(* PLC project Generated.project, CODESYS CODESYS V3.5 SP19 Patch 1 *)
(* stored: creationDateTime 2026-09-06T13:00:42.508254, modificationDateTime 2026-09-06T13:00:42.508254 *)

(* ═══════════════════════════════════════════════════════════════ ↔️ ST_TranslationHMI — Données d'échange IHM pour le Translation M3 ─────────────────────────────────────────────────────────────── 🎨 Destiné à l'affichage des états, commandes et diagnostics du translation. 📄 Structuration en Cmd / State / Safety / Bypass / Test — doc métier : DOC/AF/AF_Partie-11_Fonction_Translation_v2.3.md ═══════════════════════════════════════════════════════════════ *)
TYPE ST_TranslationHMI : STRUCT
  Cmd : ST_TranslationCmd;  (* 🎮 Commandes opérateur (manuel / maintenance) *)
  State : ST_TranslationState;  (* 🚦 États & diagnostics *)
  Cfg : ST_TranslationCfg;  (* Configurations et limites — champ Cfg manquait initialement (contrairement à ST_WinchHMI) *)
  Bypass : ST_BypassTranslation;  (* Bypass maintenance *)
  Safety : ST_SafetyTranslation;  (* 🛡️ Sécurité (FB_Safety_Translation) *)
END_STRUCT;
END_TYPE

(* ═══════════════════════════════════════════════════════════════ ST_BypassTranslation — Bypass maintenance dédiés à Translation M3 ─────────────────────────────────────────────────────────────── 🔒 Doctrine : actionnable UNIQUEMENT en MAINT_N2, RETAIN, jamais masque les autres défauts du même bloc (voir REGISTRE_ACTIONS_Bypass_v1.0 (archive)). ═══════════════════════════════════════════════════════════════ *)
TYPE ST_BypassTranslation : STRUCT
  OperatorComm : BOOL;  (* 📡 1. Communication & Systèmes auxiliaires 📡 Bypass communication esclave CANopen Joystick / heartbeat IHM *)
  DriveComm : BOOL;  (* 📡 Bypass diagnostic esclave EtherCAT AC600 (variateur) *)
  ContactorFeedback : BOOL;  (* 🔌 Bypass feedbacks contacteur de frein *)
  PhaseRotation : BOOL;  (* ⚡ Bypass défaut rotation de phases (commun machine) *)
  BrakeThermal : BOOL;  (* 🌡️ Bypass surchauffe thermique frein (commun machine) *)
  LimitSwitch : BOOL;  (* 🚧 2. Limites physiques et Positionnement 🚧 Bypass fins de course physiques avant/arrière *)
  SensorIncoherent : BOOL;  (* 🧭 Bypass incohérence mot capteurs de position *)
  MinHeight : BOOL;  (* : Bypass interlock hauteur mini M1/M2 requise pour translation *)
  MecaA : BOOL;  (* ⚙️ 3. Sécurité Mécanique (Méca A-B) 🔄 Bypass Méca A : mouvement non commandé à l'arrêt *)
  MecaB : BOOL;  (* 🛑 Bypass Méca B : absence confirmation arrêt (frein/contacteurs) *)
  Safety : BOOL;  (* 🛡️ 4. Hiérarchie & Restauration 🛡️ Bypass groupé : tous les bits qui provoquent un PowerCutOff *)
  Process : BOOL;  (* ⚙️ Bypass groupé : tous les bits qui provoquent un SafeStop *)
  Global : BOOL;  (* 🌐 Bypass Global : ignore toutes les sécurités de cet axe *)
  Initialized : BOOL := FALSE;  (* Flag restauration boot dédié (défaut FALSE non ambigu, contrairement à une valeur métier) 🚦 TRUE = bypass restauré depuis GVL_BypassRetain ce boot *)
END_STRUCT;
END_TYPE

(* ═══════════════════════════════════════════════════════════════ 🛡️ ST_SafetyTranslation — Diagnostics de sécurité pour la Translation M3 ─────────────────────────────────────────────────────────────── 🎨 Destiné à l'affichage des défauts de sécurité du translation. ═══════════════════════════════════════════════════════════════ *)
TYPE ST_SafetyTranslation : STRUCT
  Error : BOOL;  (* 🛡️ Bloc sécurité (Safety) en défaut *)
  ErrorId : WORD;  (* ❌ Code bitfield du défaut de sécurité (vue LIVE) *)
  LatchedId : WORD;  (* 🕘 Vue LATCHÉE : ErrorId figé au défaut, effacé au Reset (marqueur [HISTO]) *)
  ErrorOperatorComm : BOOL;  (* 🎮 Perte communication opérateur : joystick CAN ou heartbeat IHM (bit0) *)
  ErrorDriveComm : BOOL;  (* 📡 Perte communication EtherCAT variateur (bit1) *)
  ErrorPhaseRotation : BOOL;  (* ⚡ Mauvaise rotation de phases électriques (bit2) *)
  ErrorBrakeThermal : BOOL;  (* 🌡️ Surchauffe thermique frein commun (bit3) *)
  ErrorMecaB : BOOL;  (* 🛑 Absence confirmation arrêt (Méca B - bit4) *)
  ErrorMecaA : BOOL;  (* 🔄 Mouvement non commandé (Méca A - bit5) *)
  ErrorLimitSwitch : BOOL;  (* 🚧 Limite extrême Translation atteinte (bit6) *)
  ErrorSensorIncoherent : BOOL;  (* 🧭 Mot capteurs M3 incohérent (bit7) *)
  SafeStop : BOOL;  (* 🛡️ Décélération de sécurité demandée *)
  PowerCutOff : BOOL;  (* 🧨 Coupure puissance demandée *)
  EffectivePermitM3_Tremie : BOOL;  (* 🟢 Permis canonique M3 vers Trémie, TRUE = autorisé *)
  EffectivePermitM3_Maintenance : BOOL;  (* 🟢 Permis canonique M3 vers Maintenance/P1, TRUE = autorisé *)
  BlockedBySafety : BOOL;  (* 🚫 Synthèse globale : translation bloquée par la sécurité *)
  PowerCutOffSafety : BOOL;  (* 🧨 Synthèse sécurités critiques entraînant une coupure puissance *)
  SafeStopSafety : BOOL;  (* 🛡️ Synthèse défauts entraînant un SafeStop / Rampe rapide *)
END_STRUCT;
END_TYPE

(* ═══════════════════════════════════════════════════════════════ ST_TranslationCfg — Configurations et paramètres réglables pour Translation M3 ─────────────────────────────────────────────────────────────── 🎨 Destiné au paramétrage depuis l'IHM (RETAIN) — même patron que ST_WinchCfg. 📄 Vitesses de ralentissement d'approche réglables depuis l'IHM (RETAIN), même patron que ST_WinchCfg. ═══════════════════════════════════════════════════════════════ *)
TYPE ST_TranslationCfg : STRUCT
  CfgApproachSpeedTremie_Hz : REAL := 20;  (* 🐢 Vitesse réduite d'approche Trémie (Hz), déclenchée par capteur PV, Direction=1 — reglage nominal confirme operateur *)
  CfgApproachSpeedMaintenance_Hz : REAL := 20;  (* 🐢 Vitesse réduite d'approche Maintenance (Hz), déclenchée par capteur P1, Direction=-1 — reglage nominal confirme operateur *)
  CfgApproachSpeedP1_Hz : REAL := 20;  (* 🐢 Vitesse réduite d'approche P1 (Hz), déclenchée par capteur P2, Direction=-1 — reglage nominal confirme operateur *)
  Initialized : BOOL := FALSE;  (* Flag restauration boot (défaut FALSE non ambigu) — même patron que ST_WinchCfg 🚦 TRUE = config restaurée depuis GVL_PERSISTENT ce boot *)
END_STRUCT;
END_TYPE

(* ═══════════════════════════════════════════════════════════════ 🎮 ST_TranslationCmd — Commandes IHM pour la Translation M3 ─────────────────────────────────────────────────────────────── 🎨 Destiné au pilotage de la translation M3 depuis l'IHM. 📄 : Initialized protège SetFreq_Hz (seul réglage à survivre au reboot), sans pont générique pour ne jamais persister BtnTremie/BtnMaintenance. ═══════════════════════════════════════════════════════════════ *)
TYPE ST_TranslationCmd : STRUCT
  SelPositioning : BOOL;  (* 🎯 TRUE = positionneur sur SelTarget ; FALSE = jog libre *)
  SelTarget : INT;  (* 🔢 Numéro de la cible de position sélectionnée *)
  BtnTremie : BOOL;  (* ↔️ Requête marche vers Trémie (ex-BtnFwd), pilotage IHM exclusif *)
  BtnMaintenance : BOOL;  (* ↔️ Requête marche vers Maintenance (ex-BtnRev), pilotage IHM exclusif *)
  SetFreq_Hz : REAL;  (* 🎯 Consigne fréquence manuelle [Hz], limitée par PRG_06_Outputs *)
  InvertDirection : BOOL;  (* 🔀 Switch machine unique : GVL_IHM.Modes.Cmd.TglJoystickMaster (ST_ModesCmd), applicable à M1/M2 ET M3. 🔄 TRUE = inverse Fwd→Maintenance / Rev→Trémie (mise en service) *)
  TglMaintenanceZoneAccess : BOOL;  (* : autorisation CONSCIENTE zone Maintenance, EN PLUS de MAINT_N2 (Auth.MaintenanceM3TargetEnable) *)
  TglAllowWinchMoveAtTremie : BOOL;  (* T249 : autorisation CONSCIENTE montee/descente treuil couple (WinchSel=0) a la Tremie, EN PLUS de la garde WinchSel=2 forcee (FB_Modes) *)
  Initialized : BOOL := FALSE;  (* 🚦 TRUE = SetFreq_Hz restauré depuis GVL_PERSISTENT ce boot *)
  BtnSetAtP1 : BOOL;  (* 🎯 Forcage position P1 depuis IHM en MAINT_N2 (mise en service) *)
END_STRUCT;
END_TYPE

(* ═══════════════════════════════════════════════════════════════ 🚦 ST_TranslationState — États et retours IHM pour la Translation M3 ─────────────────────────────────────────────────────────────── 🎨 Destiné à l'affichage des retours et mesures de la translation M3. ═══════════════════════════════════════════════════════════════ *)
TYPE ST_TranslationState : STRUCT
  FBState : E_State;  (* 🚦 États & diagnostics FB_Translation 🤖 État de l'automate interne (FB_Translation) *)
  AxisBlockReason : E_TranslationTraceBlockReason;  (* 🧩 Cause prioritaire de blocage (miroir de TranslationTrace.BlockReason) *)
  Ready : BOOL;  (* 🟢 Translation prêt à fonctionner *)
  Busy : BOOL;  (* ⚙️ Mouvement en cours *)
  Done : BOOL;  (* ✅ Mouvement terminé avec succès *)
  Error : BOOL;  (* Translation en défaut *)
  ErrorId : WORD;  (* ❌ Code du défaut actif *)
  BrakeCmd : BOOL;  (* 🔓 Commande de desserrage du frein (lecture seule, TRUE = desserré) *)
  BrakeFeedback : BOOL;  (* 🔌 Retour physique direct : TRUE = frein OUVERT (desserré) *)
  PositionSensorTarget : BOOL;  (* 🎯 Capteur de détection de la position cible atteint *)
  PositionReached : BOOL;  (* ✅ Positionneur : cible sélectionnée atteinte (non mémorisé) *)
  DriveActualFreq_Hz : REAL;  (* 📈 Fréquence de sortie réelle du variateur (Hz) *)
  DriveControlWord : WORD;  (* ⚙️ Mot de commande AC600 réellement appliqué *)
  DriveFreqCmd_Hz : REAL;  (* 🎯 Commande fréquence réellement appliquée *)
  ActiveTremie : BOOL;  (* ↔️ Commande active vers Trémie *)
  ActiveMaintenance : BOOL;  (* ↔️ Commande active vers Maintenance *)
  SpeedCmd_Pct : REAL;  (* 📊 Commande active après arbitrage (0.0 à 100.0 %) *)
  FinalInterlockState : E_State;  (* 🛡️ État final lecture seule *)
  FinalInterlockReason : E_TranslationFinalInterlockReason;  (* 🛡️ Cause finale mémorisée *)
  FinalInterlockError : BOOL;  (* 🛡️ Défaut final mémorisé *)
  FinalInterlockErrorId : WORD;  (* 🛡️ Bitfield final *)
  BrakeCommandOpenConfirmed : BOOL;  (* 🔌 Contacteur/bobine desserrage confirmé, pas frein mécanique *)
  FinalBrakeTimeoutElapsed : TIME;  (* ⏱️ Écoulé watchdog 500ms *)
  DriveCommReady : BOOL;  (* 🔌 Diagnostic variateur EtherCAT (décodé — pas de bit-masking côté IHM) 📡 Variateur M3 : communication prête (StatusWord bit7) *)
  DrivePowerReady : BOOL;  (* ⚡ Variateur M3 : puissance prête (StatusWord bit0) *)
  PositionTremie : BOOL;  (* 📍 Mot capteurs et positions Translation M3 *)
  PositionPV : BOOL;
  PositionP2 : BOOL;
  PositionP1 : BOOL;
  PositionMaintenance : BOOL;
  AtTremie : BOOL;  (* : mot EXACT — front franc arrivée/cible (voir PositionXxx ci-dessus = cumulatif zone, réservé ralentissement) jeton "dernier capteur franchi" (front + libération sur mouvement confirmé) — logique de positionnement *)
  AtPV : BOOL;
  AtP2 : BOOL;
  AtP1 : BOOL;
  AtMaintenance : BOOL;
  M3StatusText : STRING(80);  (* T249-B : texte statut position M3 (INFO, lecture seule) — jeton "at position" sur front capteur sinon zone SensorsWord. Ex "M3 a P1 -> Maintenance", "M3 entre P2 et P1" *)
  EstimatedPosM3_M : REAL;  (* 📏 Position continue estimée en mètres (0.0 m Maint -> +X m Trémie) — persistante, survit reboot *)
  SensorsWord : BYTE;  (* bit4=Trémie, bit3=PV, bit2=P2, bit1=P1, bit0=Maintenance *)
  SensorWordIncoherent : BOOL;
  LimitSwitchTremie : BOOL;  (* 🚧 Fin de course extrême Trémie (ex-LimitSwitchFwd) *)
  LimitSwitchMaintenance : BOOL;  (* 🚧 Fin de course extrême Maintenance (ex-LimitSwitchRev) *)
  DriveThermalOk : BOOL;  (* Retour disjoncteur thermique moteur/variateur AC600 — diagnostic seul, l'AC600 se protège lui-même *)
  MaintenanceTargetEnable : BOOL;  (* 🔓 TRUE = Autorise le déplacement vers la cible 4 (Maintenance) ; actif uniquement en mode MAINT_N2 *)
  SimulationModeActive : BOOL;
  HeightInterlockBlocking : BOOL;  (* : TRUE = translation bloquée, M1 ou M2 sous la hauteur mini requise *)
  OdometryGainActive : REAL;  (* 📏 T301 — Odométrie M3 : gain actif + mesure PROPOSÉE P2 <-> PV (jamais appliquée, recopie manuelle) Gain consommé par l'estimateur, m/(Hz.s) *)
  OdometryCalibValid : BOOL;  (* TRUE = gain calculé depuis le réglage Calib* (défaut 2,0 s compris) ; FALSE = gain de repli *)
  OdometryMeasureActive : BOOL;  (* Mesure P2 <-> PV en cours *)
  OdometryMeasuredTime_S : REAL;  (* Dernier temps mesuré P2 <-> PV (s) -> à recopier dans _TranslationCalibTimeP2PV_S *)
  OdometryMeasuredFreqAvg_Hz : REAL;  (* Fréquence moyenne de la mesure (Hz) -> à recopier dans _TranslationCalibFreq_Hz *)
  OdometryMeasuredFreqSpread_Hz : REAL;  (* Écart max - min de fréquence : petit = vitesse constante, mesure fiable *)
  OdometryMeasuredGain : REAL;  (* Gain qui résulterait de la mesure, m/(Hz.s) *)
  OdometryMeasureCount : UDINT;  (* Nombre de mesures abouties depuis le démarrage *)
END_STRUCT;
END_TYPE

(* values of E_State: DISABLED: Enable faux, neutralisé; INIT: Démarrage / vérifs; READY: Prêt, attend ordre; BUSY: Action en cours; DONE: Action terminée; STOPPING: Décél rampe avant arrêt (StartStop=FALSE ou SafeStop=TRUE); ERROR: Défaut actif non acquitté (FB en erreur — HMI non aveugle) *)

{attribute 'qualified_only'}
{attribute 'strict'}
TYPE E_State : (DISABLED := 0, INIT := 1, READY := 2, BUSY := 3, DONE := 4, STOPPING := 5, ERROR := 6);
END_TYPE

{attribute 'qualified_only'}
{attribute 'strict'}
TYPE E_TranslationFinalInterlockReason : (NONE := 0, BRAKE_COMMAND_NOT_CONFIRMED := 1, RESTART_INHIBITED := 2);
END_TYPE

(* values of E_TranslationTraceBlockReason: NONE: ✅ Aucun blocage — permis de mouvement effectif; POWER_CUTOFF: 🧨 Coupure puissance amont (instSafetyTranslationM3.PowerCutOff) — priorité max; SAFESTOP: 🟧 SafeStop effectif (InputModule OR safety M3); SAFETY_FAULT: 🛡️ Défaut safety M3 latched (FB_Safety_Translation.Fault.Error); HEIGHT_INTERLOCK: 🚧 Interlock hauteur M1/M2 actif (risque collision); DRIVE_UNAVAILABLE: 📡 Variateur AC600 injoignable / non opérationnel; FINAL_INTERLOCK: 🛑 Barrière finale en défaut (frein / redémarrage); FAULT: ❌ Défaut mouvement M3 latched (FB_Translation.Fault.Error) *)

{attribute 'qualified_only'}
{attribute 'strict'}
TYPE E_TranslationTraceBlockReason : (NONE := 0, POWER_CUTOFF := 1, SAFESTOP := 2, SAFETY_FAULT := 3, HEIGHT_INTERLOCK := 4, DRIVE_UNAVAILABLE := 5, FINAL_INTERLOCK := 6, FAULT := 7);
END_TYPE
